PROGRAM MAIN
VAR
	stEmployee : ST_Employee;
	nStEmployeeElementCount : ULINT;
	fbCountStructElements : FB_CountStructElements;
END_VAR

fbCountStructElements(stAny := stEmployee, nElementsCount=> nStEmployeeElementCount );

END_PROGRAM

(* stored: Version 1.1.0.1, ProductVersion 3.1.4024.11
   POU MAIN: Id {49ba8e01-0aaf-45d2-ab7f-4d1bdf3fd475}, SpecialFunc None *)
